{attribute 'qualified_only'}
VAR_GLOBAL

END_VAR

(* stored: Version 1.1.0.1, ProductVersion 3.1.4020.6
   GVL GVL: Id {cb054416-d49d-4893-9f08-75335226c7c7} *)
